FUNCTION_BLOCK ABSTRACT ContinuousDrive EXTENDS Drive

METHOD ABSTRACT moveContinuous : BOOL
VAR_INPUT
	direction : MC_Direction;
END_VAR
END_METHOD

END_FUNCTION_BLOCK

(* stored: Version 1.1.0.1, ProductVersion 3.1.4024.11
   POU ContinuousDrive: Id {cae9604f-13b9-413a-a13e-3ee322a28517}, SpecialFunc None
   Method moveContinuous: Id {9368f197-cd84-4fc5-91f0-a34190040adf} *)
